VAR_GLOBAL // STATE
    g_inp: DINT;
    p_b: BOOL;
    p_x: DINT;
    p_y: LREAL;
    p_ve: g_E;
    p_v1: DINT;
    p_v2: TupleStruct;
    p_v3: TupleStruct__1;
    p_tv: TupleStruct__2;
    p_j: DINT;
    p_r: LREAL;
    p: p_location;
END_VAR

(* stored: ProductVersion 3.1.0.18, Version 1.1.0.1 *)
